KUKA KRL data list: Up21.dat

&ACCESS RVO1
&REL 158
&COMMENT VW380 HO_Behaelter_links
&PARAM EDITMASK = Up999[1-999]
&PARAM TPVW_VERSION = 8.3.18
&PARAM TEMPLATE = C:\KRC\Roboter\Template\upvorgabe
&PARAM DISKPATH = UPs
DEFDAT UP21
; FOLD ;%{H} %MKUKATPVW
; ENDFOLD
; interface to basic routines
 EXT  BAS (BAS_COMMAND  :IN,REAL  :IN )
; interface to VW-standard routines
EXT VW (VW_COMMAND:IN, BOOL: IN, REAL:IN, REAL:IN, REAL:IN, REAL:IN, BOOL :IN, E6POS :IN )
; interface to VW_USER - Call
EXT  VW_USER (VW_USER_CMD :IN,INT :IN,REAL  :IN,REAL  :IN,REAL  :IN,REAL  :IN,REAL  :IN,REAL  :IN,REAL  :IN,REAL  :IN,REAL  :IN,BOOL  :IN)
EXT  VW_USR_R (VW_USER_CMD :IN,INT :IN,REAL  :IN,REAL  :IN,REAL  :IN,REAL  :IN,REAL  :IN,REAL  :IN,REAL  :IN,REAL  :IN,REAL  :IN,BOOL  :IN)
EXT  IBGN (IBGN_COMMAND  :IN,BOOL  :IN,REAL  :IN,REAL  :IN,BOOL  :IN,E6POS  :OUT )
; interface select routine
EXTFCT INT  SELECT (SUBTYPE  :IN,INT  :IN,BOOL  :IN,ARI_TYP  :IN,INT  :IN,BOOL_TYP  :IN,INT  :IN,BOOL  :IN)
INT VW_NEXT_FREE = 22
INT VW_NFREE_SPS = 22
INT VW_MAX_SPS = 122
DECL VW_MPARA_TYP P1_D = {TOOL_NO 11,BASE_NO 0,VB 100,VE 0,ACC 100,TRG_TIME 0,MOVE_TYPE #PTP_MOTION}
DECL E6POS P1 = {X 556.5872, Y 1169.977, Z 573.7128, A 30.0, B -0.000000112, C -180.0, S 2, T 3 , E1 0.0, E2 0.0, E3 0.0, E4 0.0, E5 0.0, E6 0.0}
DECL VW_MPARA_TYP P2_D = {TOOL_NO 11,BASE_NO 0,VB 100,VE 100,ACC 100,TRG_TIME 0,MOVE_TYPE #PTP_MOTION}
DECL E6POS P2 = {X 556.5872, Y 1169.977, Z 573.7128, A 30.0, B -0.000000112, C -180.0, S 2, T 3 , E1 0.0, E2 0.0, E3 0.0, E4 0.0, E5 0.0, E6 0.0}
DECL VW_MPARA_TYP P3_D = {TOOL_NO 11,BASE_NO 0,VB 250,VE 50,ACC 100,TRG_TIME 0,MOVE_TYPE #GLUE_MOTION}
DECL E6POS P3 = {X 534.301, Y 1168.777, Z 569.688, A 30.0, B -0.000000111, C -180.0, S 2, T 3 , E1 0.0, E2 0.0, E3 0.0, E4 0.0, E5 0.0, E6 0.0}
DECL VW_MPARA_TYP P4_D = {TOOL_NO 11,BASE_NO 0,VB 250,VE 50,ACC 50,TRG_TIME 0,MOVE_TYPE #GLUE_MOTION}
DECL E6POS P4 = {X 491.0204, Y 1166.447, Z 561.8719, A 30.0, B -0.000000109, C -180.0, S 2, T 3 , E1 0.0, E2 0.0, E3 0.0, E4 0.0, E5 0.0, E6 0.0}
DECL VW_MPARA_TYP P5_D = {TOOL_NO 11,BASE_NO 0,VB 250,VE 50,ACC 100,TRG_TIME 0,MOVE_TYPE #GLUE_MOTION}
DECL E6POS P5 = {X 384.2884, Y 1184.738, Z 561.8702, A 30.0, B -0.000000115, C -180.0, S 2, T 3 , E1 0.0, E2 0.0, E3 0.0, E4 0.0, E5 0.0, E6 0.0}
DECL VW_MPARA_TYP P6_D = {TOOL_NO 11,BASE_NO 0,VB 100,VE 100,ACC 100,TRG_TIME 0,MOVE_TYPE #PTP_MOTION}
DECL E6POS P6 = {X 384.2884, Y 1184.738, Z 579.3517, A 30.0, B -0.000000117, C -180.0, S 2, T 3 , E1 0.0, E2 0.0, E3 0.0, E4 0.0, E5 0.0, E6 0.0}
DECL VW_MPARA_TYP P7_D = {TOOL_NO 11,BASE_NO 0,VB 100,VE 100,ACC 100,TRG_TIME 0,MOVE_TYPE #PTP_MOTION}
DECL E6POS P7 = {X 442.7902, Y 1762.65, Z 1887.477, A 21.55133, B 0.189589, C -113.1255, S 2, T 11 , E1 0.0, E2 0.0, E3 0.0, E4 0.0, E5 0.0, E6 0.0}
DECL VW_MPARA_TYP P8_D = {TOOL_NO 11,BASE_NO 0,VB 100,VE 100,ACC 100,TRG_TIME 0,MOVE_TYPE #PTP_MOTION}
DECL E6POS P8 = {X 1530.675, Y -755.5926, Z 1810.376, A -61.04628, B -10.65187, C -125.4632, S 2, T 10 , E1 0.0, E2 0.0, E3 0.0, E4 0.0, E5 0.0, E6 0.0}
DECL VW_MPARA_TYP P9_D = {TOOL_NO 11,BASE_NO 0,VB 100,VE 100,ACC 100,TRG_TIME 0,MOVE_TYPE #PTP_MOTION}
DECL E6POS P9 = {X 591.5993, Y -1509.546, Z 1783.347, A -93.98762, B -12.54844, C -129.5027, S 2, T 10 , E1 0.0, E2 0.0, E3 0.0, E4 0.0, E5 0.0, E6 0.0}
DECL VW_MPARA_TYP P10_D = {TOOL_NO 11,BASE_NO 0,VB 100,VE 100,ACC 100,TRG_TIME 0,MOVE_TYPE #PTP_MOTION}
DECL E6POS P10 = {X 877.1592, Y -1069.184, Z 454.6454, A -24.41104, B -1.433861, C -174.7075, S 2, T 10 , E1 0.0, E2 0.0, E3 0.0, E4 0.0, E5 0.0, E6 0.0}
DECL VW_MPARA_TYP P11_D = {TOOL_NO 11,BASE_NO 0,VB 100,VE 0,ACC 100,TRG_TIME 0,MOVE_TYPE #PTP_MOTION}
DECL E6POS P11 = {X 824.3167, Y -1052.805, Z -33.54369, A 2.361682, B 4.729669, C 179.8833, S 2, T 2 , E1 0.0, E2 0.0, E3 0.0, E4 0.0, E5 0.0, E6 0.0}
DECL VW_MPARA_TYP P12_D = {TOOL_NO 11,BASE_NO 3,VB 400,VE 0,ACC 100,TRG_TIME 0,MOVE_TYPE #PATH_MOTION}
DECL E6POS P12 = {X 814.3167, Y -1062.805, Z -43.54369, A 2.361682, B 4.729669, C 179.8833, S 2, T 2 , E1 0.0, E2 0.0, E3 0.0, E4 0.0, E5 0.0, E6 0.0}
DECL VW_MPARA_TYP P13_D = {TOOL_NO 11,BASE_NO 3,VB 400,VE 0,ACC 100,TRG_TIME 0,MOVE_TYPE #PATH_MOTION}
DECL E6POS P13 = {X 2089.785, Y -1054.905, Z -43.54038, A 2.361682, B 4.729669, C 179.8833, S 2, T 2 , E1 0.0, E2 0.0, E3 0.0, E4 0.0, E5 0.0, E6 0.0}
DECL VW_MPARA_TYP P14_D = {TOOL_NO 11,BASE_NO 31,VB 50,VE 100,ACC 100,TRG_TIME 5,MOVE_TYPE #PATH_MOTION}
DECL E6POS P14 = {X 3.930478, Y -0.000027, Z -2.938142, A 0.0, B 0.0, C 0.0, S 2, T 2 , E1 0.0, E2 0.0, E3 0.0, E4 0.0, E5 0.0, E6 0.0}
DECL VW_MPARA_TYP P15_D = {TOOL_NO 11,BASE_NO 31,VB 400,VE 100,ACC 100,TRG_TIME 0,MOVE_TYPE #PATH_MOTION}
DECL E6POS P15 = {X 5.282126, Y 0.000001, Z -72.19976, A 0.0, B 0.0, C 0.0, S 2, T 2 , E1 0.0, E2 0.0, E3 0.0, E4 0.0, E5 0.0, E6 0.0}
DECL VW_MPARA_TYP P16_D = {TOOL_NO 11,BASE_NO 31,VB 400,VE 100,ACC 100,TRG_TIME 0,MOVE_TYPE #PATH_MOTION}
DECL E6POS P16 = {X -98.53275, Y -20.71485, Z -72.19978, A -9.969234, B 0.0, C 0.0, S 2, T 2 , E1 0.0, E2 0.0, E3 0.0, E4 0.0, E5 0.0, E6 0.0}
DECL VW_MPARA_TYP P17_D = {TOOL_NO 11,BASE_NO 31,VB 400,VE 100,ACC 100,TRG_TIME 0,MOVE_TYPE #PATH_MOTION}
DECL E6POS P17 = {X -98.01331, Y -17.21537, Z -72.35353, A -11.34339, B -0.078733, C -3.28507, S 2, T 2 , E1 0.0, E2 0.0, E3 0.0, E4 0.0, E5 0.0, E6 0.0}
DECL VW_MPARA_TYP P18_D = {TOOL_NO 11,BASE_NO 0,VB 1500,VE 0,ACC 100,TRG_TIME 0,MOVE_TYPE #PATH_MOTION}
DECL E6POS P18 = {X 944.9223, Y -1048.387, Z 46.61262, A 13.7443, B 4.73875, C 177.5329, S 2, T 2 , E1 0.0, E2 0.0, E3 0.0, E4 0.0, E5 0.0, E6 0.0}
DECL VW_MPARA_TYP P19_D = {TOOL_NO 11,BASE_NO 0,VB 100,VE 100,ACC 100,TRG_TIME 0,MOVE_TYPE #PTP_MOTION}
DECL E6POS P19 = {X 824.3167, Y -1052.805, Z 57.00082, A 2.361682, B 4.729669, C 179.8833, S 2, T 2 , E1 0.0, E2 0.0, E3 0.0, E4 0.0, E5 0.0, E6 0.0}
DECL VW_MPARA_TYP P20_D = {TOOL_NO 11,BASE_NO 0,VB 100,VE 100,ACC 100,TRG_TIME 0,MOVE_TYPE #PTP_MOTION}
DECL E6POS P20 = {X 865.1878, Y -1042.062, Z 803.3944, A 3.272736, B 3.014662, C 179.9311, S 2, T 2 , E1 0.0, E2 0.0, E3 0.0, E4 0.0, E5 0.0, E6 0.0}
DECL VW_MPARA_TYP P21_D = {TOOL_NO 11,BASE_NO 0,VB 100,VE 0,ACC 100,TRG_TIME 0,MOVE_TYPE #PTP_MOTION}
DECL E6POS P21 = {X 856.7742, Y -895.0887, Z 803.2177, A 3.272736, B 3.014662, C 179.9311, S 2, T 2 , E1 0.0, E2 0.0, E3 0.0, E4 0.0, E5 0.0, E6 0.0}
ENDDAT
